INTERFACE ITF_Analogue

METHOD GetValue : INT
VAR_INPUT
END_VAR
END_METHOD

END_INTERFACE

(* stored: Version 1.1.0.1, ProductVersion 3.1.4024.12
   Itf ITF_Analogue: Id {1c3863cb-38a1-42ec-a973-3d7f7caf3fb0}
   Method GetValue: Id {8a25bba1-0ec8-49bd-a615-831e194b3e56} *)
